{attribute 'linkalways'} 
{attribute 'no_explicit_call' := 'This FB is a CLASS and must be accessed using methods or properties'}
{attribute 'enable_dynamic_creation'}
FUNCTION_BLOCK _ETcVnNbc EXTENDS EnumDatatypeBase
VAR
	localData : ETcVnNbc;
	activeData : REFERENCE TO ETcVnNbc;
	enumBaseDatatype : _UDINT(localData);
END_VAR

METHOD PRIVATE AddLocalEnumeration
VAR_INPUT
	Enumeration : T_MAXSTRING;
	Value : ETcVnNbc;
END_VAR
AddEnumeration(Enumeration, Value);
END_METHOD

PROPERTY PUBLIC Address : PVOID
GET
Address := ADR(activeData);
END_GET
END_PROPERTY

METHOD PUBLIC ClearReference
VAR_INPUT
END_VAR
activeData REF= localData;
SetBaseDatatypeReference();
END_METHOD

METHOD PUBLIC Clone : I_Datatype
VAR
    pClone : POINTER TO _ETcVnNbc;
END_VAR
pClone := __NEW(_ETcVnNbc(InitialValue := Value));
Clone := pClone^;
END_METHOD

METHOD FB_init : BOOL
VAR_INPUT
	bInitRetains : BOOL; // if TRUE, the retain variables are initialized (warm start / cold start)
	bInCopyCode : BOOL;  // if TRUE, the instance afterwards gets moved into the copy code (online change)
	InitialValue : ETcVnNbc;
END_VAR
localData := InitialValue;
AddBaseDatatype(enumBaseDatatype);
ClearReference();

AddLocalEnumeration('TCVN_NBC_CLASSIFIER', ETcVnNbc.TCVN_NBC_CLASSIFIER);
AddLocalEnumeration('TCVN_NBC_NOVELTY_DETECTOR', ETcVnNbc.TCVN_NBC_NOVELTY_DETECTOR);
END_METHOD

PROPERTY PUBLIC Identifier : T_MAXSTRING
GET
Identifier := 'ETcVnNbc';
END_GET
END_PROPERTY

METHOD IsEnumeratorValueEqual : BOOL
VAR_INPUT
	Enumerator : I_KeyValueForwardEnumerator;
END_VAR
VAR
	storedValue : ETcVnNbc;
END_VAR
IF NOT Enumerator.TryGet(storedValue) THEN
	RETURN;
END_IF

IsEnumeratorValueEqual := storedValue = activeData;
END_METHOD

METHOD PUBLIC MakeReferenceTo
VAR_INPUT
	ReferenceTarget : REFERENCE TO ETcVnNbc;
END_VAR
activeData REF= ReferenceTarget;
SetBaseDatatypeReference();
END_METHOD

METHOD PROTECTED SetBaseDatatypeReference
VAR_INPUT
END_VAR
enumBaseDatatype.MakeReferenceTo(activeData);
END_METHOD

PROPERTY PUBLIC Size : UDINT
GET
Size := SIZEOF(activeData);
END_GET
END_PROPERTY

METHOD TryMakeReferenceTo : BOOL
VAR_INPUT
	Target : I_Datatype;
END_VAR
VAR
	targetAsEnum : I_EnumDatatype;
	pTargetData : POINTER TO ETcVnNbc;
END_VAR
IF NOT Target.TryResolveAsEnumDatatype(targetAsEnum) THEN
	RETURN;
END_IF

IF targetAsEnum.Identifier <> Identifier THEN
	RETURN;
END_IF

pTargetData := Target.Address;
activeData REF= pTargetData^;
SetBaseDatatypeReference();
TryMakeReferenceTo := TRUE;
END_METHOD

PROPERTY PUBLIC Value : ETcVnNbc
GET
Value := activeData;
END_GET
SET
activeData := Value;
END_SET
END_PROPERTY

END_FUNCTION_BLOCK

(* stored: Version 1.1.0.1
   POU _ETcVnNbc: Id {874df502-9ad7-44ef-b6d6-af68b2feea80}, SpecialFunc None
   Folder Constructor: Id {2a258ec7-e3f6-4f8a-a3a4-6efec3c3cb40}
   Folder Private: Id {11871fa5-405d-4ca4-bdd7-90c0815adc0c}
   Folder Protected: Id {f4d08b99-3d0b-4b98-917b-8892a68d7c67}
   Method AddLocalEnumeration: Id {dc82133f-1782-443f-abb9-59e7a5c37002}
   Property Address: Id {90d47084-423a-4992-8758-826c1d5fce7c}
   Get Get: Id {d9fa7176-495e-420a-b982-166c5679f378}
   Method ClearReference: Id {210ec23a-c31d-434a-9d4a-ffe2b34d5e76}
   Method Clone: Id {c084db4c-52bb-4b24-93b2-5b19b3a11674}
   Method FB_init: Id {c31b8f2e-51df-47c0-8e3f-bebd783d3501}
   Property Identifier: Id {8c9344ed-9274-4a8e-9f6e-12ffd552f967}
   Get Get: Id {fa98e414-f81e-4b97-9aea-39110bb449d0}
   Method IsEnumeratorValueEqual: Id {b2cd882a-862b-4531-b974-fe676a7708ed}
   Method MakeReferenceTo: Id {215c0edd-bf00-4a2a-8920-a7299853335d}
   Method SetBaseDatatypeReference: Id {11c75327-d73f-4e19-a920-3bfda06f4ce8}
   Property Size: Id {a92805a4-cd99-4b97-b7cd-9e64b75bcd17}
   Get Get: Id {fbea3e7e-6a44-457c-a570-4c49c1cdd3f0}
   Method TryMakeReferenceTo: Id {dffdff54-dbe5-496b-86ec-2752e5f2701b}
   Property Value: Id {30811ff2-46e0-473c-bf92-318ae77e9f8c}
   Get Get: Id {99fe13d2-c3c5-4f46-bcc1-412f28b68b46}
   Set Set: Id {bb7b6ffc-9896-4b1a-9455-770da9d60792} *)
